INTERFACE ITF_Valve

PROPERTY ActualState : E_ValveState
GET
END_GET
END_PROPERTY

METHOD Close : BOOL
VAR_INPUT
END_VAR
END_METHOD

PROPERTY EmergencyStatus : BOOL
GET
END_GET
END_PROPERTY

METHOD Open : BOOL
VAR_INPUT
END_VAR
END_METHOD

PROPERTY OperatingMode : BOOL
GET
END_GET
END_PROPERTY

METHOD Reset : BOOL
VAR_INPUT
END_VAR
END_METHOD

METHOD SetMode : BOOL
VAR_INPUT
END_VAR
END_METHOD

END_INTERFACE

(* stored: Version 1.1.0.1, ProductVersion 3.1.4024.12
   Itf ITF_Valve: Id {23478fd0-4917-4f3c-bacd-f8f2c3e8833e}
   Folder Methods: Id {baddf355-ae32-47ad-aef2-70ca23b070fe}
   Folder Properties: Id {6d9d25d0-e5b0-4a9d-901c-e738470977aa}
   Property ActualState: Id {4048e3cf-1901-4fb0-b3e3-cadad5461c50}
   Get Get: Id {76a718e2-a1cd-4ce2-a1ef-9dca22eb67a3}
   Method Close: Id {52142592-4b90-4cfe-8148-6fb6e4af0466}
   Property EmergencyStatus: Id {c4fefea5-9dd9-44f2-9f49-b820e3cf5062}
   Get Get: Id {a6311909-e883-4491-b0c2-e6635f50e2c0}
   Method Open: Id {ca3aff26-be70-4831-a91e-e48cf7ecea28}
   Property OperatingMode: Id {aec482d6-a14b-4c1d-9656-4ab670725f10}
   Get Get: Id {e75f3792-5240-4fed-b756-fb81f3f8e57b}
   Method Reset: Id {07d4e633-d21f-47cd-b574-f7ddd71de663}
   Method SetMode: Id {c3f27805-b695-4c09-ab53-43ef7802b59d} *)
